(* IEC 61131-3 sources: Word/plc-course/08-counters/labs/starter, 3 files *)

(* ---- 08-1-bottle-packing.st ---- *)
(* Lab 08-1: Bottle packing - count bottles into a box, index the full box, start again.
   Module 08 (Counters). STARTER - the declarations are done for you;
   write the logic where it says TODO, then run:
     python3 tools/plctest.py 08-counters/labs/starter/08-1-bottle-packing.st *)

PROGRAM BottlePacking
  VAR (* I/O - addresses follow the OpenPLC convention *)
    BottlePE   AT %IX0.0 : BOOL;  (* Photo-eye at the end of the infeed: TRUE while a bottle blocks the beam *)
    ResetPB    AT %IX0.1 : BOOL;  (* Count reset push-button, NO: the operator has fitted a new, empty box *)
    InfeedConv AT %QX0.0 : BOOL;  (* Infeed conveyor motor: carries bottles into the box *)
    BoxConv    AT %QX0.1 : BOOL;  (* Box conveyor motor: moves the full box out and an empty one in *)
  END_VAR
  VAR (* HMI settings and displays - part of the lab interface *)
    BoxSize     : INT := 12;      (* bottles per box, 1..48 *)
    IndexTime   : TIME := T#2s;   (* how long the box conveyor runs to index one box *)
    BottleCount : INT;            (* bottles counted into the box being filled *)
  END_VAR
  VAR RETAIN (* a production total: on a real PLC it must survive a power cut *)
    BoxesPacked : DINT;           (* full boxes; ResetPB does not touch it *)
  END_VAR
  VAR (* internal - add your own variables here: a counter, a timer,
         edge detectors ... *)
    Spare : BOOL;
  END_VAR

  (* TODO: replace these placeholders with your logic.
     - Count bottles (rising edges of BottlePE) into BottleCount.
     - When BottleCount reaches BoxSize: stop the infeed at once, run the box
       conveyor for IndexTime, add one to BoxesPacked.
     - When the index ends: count from zero again and restart the infeed.
     - ResetPB: count held at zero and infeed stopped while it is held. *)
  InfeedConv := FALSE;
  BoxConv := FALSE;
  BottleCount := 0;
END_PROGRAM

CONFIGURATION Config0
  RESOURCE Res0 ON PLC
    TASK MainTask(INTERVAL := T#10ms, PRIORITY := 0);
    PROGRAM Inst0 WITH MainTask : BottlePacking;
  END_RESOURCE
END_CONFIGURATION

(* ---- 08-2-car-park.st ---- *)
(* Lab 08-2: Car park up/down counter with capacity, FULL sign and manual preset.
   Module 08 (Counters). STARTER - the declarations are done for you;
   write the logic where it says TODO, then run:
     python3 tools/plctest.py 08-counters/labs/starter/08-2-car-park.st *)

PROGRAM CarPark
  VAR (* I/O - addresses follow the OpenPLC convention *)
    EntryLoop AT %IX0.0 : BOOL;  (* Vehicle detector, entry lane: TRUE while a car is over the loop *)
    ExitLoop  AT %IX0.1 : BOOL;  (* Vehicle detector, exit lane: TRUE while a car is over the loop *)
    PresetPB  AT %IX0.2 : BOOL;  (* Attendant's preset push-button, NO: load PresetValue into the count *)
    FullSign  AT %QX0.0 : BOOL;  (* "FULL" sign at the entrance *)
  END_VAR
  VAR (* HMI settings and displays - part of the lab interface *)
    Capacity    : INT := 50;     (* number of parking spaces *)
    PresetValue : INT;           (* cars the attendant counted by walking round *)
    SpacesFree  : INT;           (* for the "spaces" sign: never negative *)
  END_VAR
  VAR RETAIN (* the cars do not leave when the power fails *)
    CarCount    : INT;           (* cars in the car park *)
  END_VAR
  VAR (* internal - add your own variables here: edge detectors or a
         counter block ... *)
    Spare : BOOL;
  END_VAR

  (* TODO: replace these placeholders with your logic.
     - CarCount: +1 per car arriving on EntryLoop, -1 per car arriving on
       ExitLoop. Never below 0. It may go ABOVE Capacity.
     - FullSign when CarCount >= Capacity; SpacesFree never negative.
     - PresetPB loads PresetValue (negative counts as 0). *)
  CarCount := 0;
  FullSign := FALSE;
  SpacesFree := 0;
END_PROGRAM

CONFIGURATION Config0
  RESOURCE Res0 ON PLC
    TASK MainTask(INTERVAL := T#10ms, PRIORITY := 0);
    PROGRAM Inst0 WITH MainTask : CarPark;
  END_RESOURCE
END_CONFIGURATION

(* ---- 08-3-production-counts.st ---- *)
(* Lab 08-3: Production counts - good/reject counters, total, yield, shift reset.
   Module 08 (Counters). STARTER - the declarations are done for you;
   write the logic where it says TODO, then run:
     python3 tools/plctest.py 08-counters/labs/starter/08-3-production-counts.st *)

PROGRAM ProductionCounts
  VAR (* I/O - addresses follow the OpenPLC convention *)
    GoodPE       AT %IX0.0 : BOOL;  (* Photo-eye on the outfeed: TRUE while an accepted pack is in the beam *)
    RejectPE     AT %IX0.1 : BOOL;  (* Photo-eye on the reject chute: TRUE while a rejected pack passes *)
    ShiftResetPB AT %IX0.2 : BOOL;  (* Shift-change push-button, NO *)
    LowYieldLamp AT %QX0.0 : BOOL;  (* Low-yield warning lamp on the line *)
  END_VAR
  VAR (* HMI settings - part of the lab interface *)
    MinSample  : DINT := 20;        (* no yield warning until this many packs this shift *)
    YieldLimit : REAL := 95.0;      (* warn when the yield is below this, % *)
  END_VAR
  VAR RETAIN (* HMI displays that must survive a power cut *)
    GoodCount       : DINT;         (* accepted packs this shift *)
    RejectCount     : DINT;         (* rejected packs this shift *)
    LastShiftGood   : DINT;         (* snapshot taken at the last shift change *)
    LastShiftReject : DINT;
    LastShiftYield  : REAL;
    LifetimeTotal   : DINT;         (* every pack since commissioning: no reset *)
  END_VAR
  VAR (* HMI displays, recalculated every scan *)
    TotalCount : DINT;              (* GoodCount + RejectCount *)
    YieldPct   : REAL;              (* 100 x good / total; 0.0 while the total is 0 *)
  END_VAR
  VAR (* internal - add your own variables here: edge detectors, constants ... *)
    Spare : BOOL;
  END_VAR

  (* TODO: replace these placeholders with your logic.
     - Count good packs and rejects (one per pack), and every pack into
       LifetimeTotal, which must never wrap round.
     - TotalCount and YieldPct (a REAL; 0.0 while TotalCount is 0).
     - On a PRESS of ShiftResetPB: copy the shift figures into the LastShift
       variables, then start the shift counts again from zero.
     - LowYieldLamp: at least MinSample packs AND YieldPct below YieldLimit. *)
  TotalCount := 0;
  YieldPct := 0.0;
  LowYieldLamp := FALSE;
END_PROGRAM

CONFIGURATION Config0
  RESOURCE Res0 ON PLC
    TASK MainTask(INTERVAL := T#10ms, PRIORITY := 0);
    PROGRAM Inst0 WITH MainTask : ProductionCounts;
  END_RESOURCE
END_CONFIGURATION
